VAR_GLOBAL
END_VAR

(* stored: Version 1.1.0.1, ProductVersion 3.1.4024.11
   GVL OP70_Recipe: Id {43ae45c4-2a1f-4225-9e0e-afa3bc693577} *)
